Fanuc KAREL source: RESET.kl

PROGRAM T
%NOLOCKGROUP
VAR
 v0 : BOOLEAN
BEGIN
 RESET(v0)
END T
